// TIA Portal project "PWM TEST" (V16)

(* hardware
DEVICE "S7-1200 station_1"  S7-1200 Station
   slot 0: "Rack_0"  S7-1200 Rack  Rack  V1.0
   slot 1: "PLC_1"  CPU 1214C DC/DC/DC  6ES7 214-1AG40-0XB0  V4.2
   slot 2: "AI 4x13BIT/AQ 2x14BIT_1"  6ES7 234-4HE32-0XB0  V2.1
DEVICE "HMI_1"  KTP1200 Basic DP
   slot 0: "HMI_1"  KTP1200 Basic DP  6AV2 123-2MA03-0AX0  16.0.0.0
   slot 1: "HMI_RT_1"  KTP1200 Basic DP  6AV2 123-2MA03-0AX0  16.0.0.0
   slot 7: "HMI_1.MPI/DP_CP_1"  MPI/DP Interface  16.0.0.0
*)

// ===== PLC "PLC_1"  CPU 1214C DC/DC/DC =====

VAR_GLOBAL   // PLC tag table "Default tag table"
   "SENSOR_TOP" AT %IW64 : Int;
   "SENSOR BOTTOM" AT %IW66 : Int;
   "PUMP_PWM" AT %QW98 : Int;
   "Tag_1" AT %MD4 : Real;
   "SET POINT TANK2" AT %MW12 : Int;
   "Tag_4" AT %MD6 : Real;
   "SENSOR_CENTIMETER 2" AT %MW10 : Int;
   "Tag_5" AT %MD14 : Real;
   "SENSOR_CENTIMETER 1" AT %MW16 : Int;
   "DATA MV TANK 2" AT %MD18 : Real;
   "Tag_7" AT %MW20 : Int;
END_VAR

DATA_BLOCK "Data_TCP"   // DB2
{ S7_Optimized_Access := 'FALSE' }
VERSION : 0.1
   VAR
      DATA : Array[0..5] of Int;
   END_VAR
BEGIN
END_DATA_BLOCK

DATA_BLOCK "MB_Config"   // DB3
{ S7_Optimized_Access := 'FALSE' }
VERSION : 0.1
   VAR
      CONNECT : TCON_IP_v4;
      NDR : Bool;
      DR : Bool;
      ERROR : Bool;
      STATUS : Word;
   END_VAR
BEGIN
   CONNECT.InterfaceId := 64;
   CONNECT.ID := 1;
   CONNECT.ConnectionType := 11;
   CONNECT.RemoteAddress.ADDR[1] := 192;
   CONNECT.RemoteAddress.ADDR[2] := 168;
   CONNECT.RemoteAddress.ADDR[3] := 0;
   CONNECT.RemoteAddress.ADDR[4] := 100;
   CONNECT.LocalPort := 502;
END_DATA_BLOCK

DATA_BLOCK "DATA PID"   // DB6
{ S7_Optimized_Access := 'TRUE' }
VERSION : 0.1
   VAR
      "SP TANK2" : Real;
      "MV TANK2" : Real;
      "MV TANK2 Conv" : Real;
   END_VAR
BEGIN
END_DATA_BLOCK

FUNCTION "Scale" : Void   // FC1, LAD
{ S7_Optimized_Access := 'TRUE' }
VERSION : 0.1
BEGIN

REGION Network 1: SECSOR TANK 1
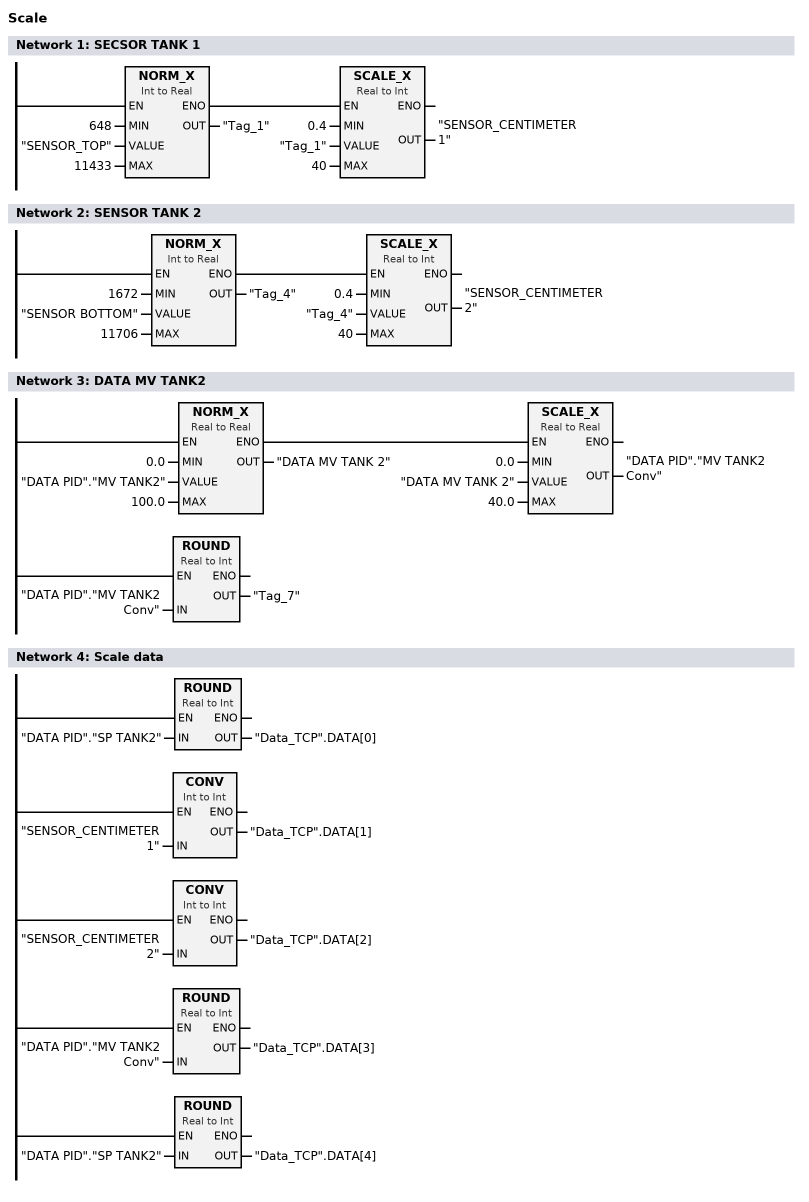
   RUNG wire#powerrail
      { S7_Templates := "[SrcType := Int, DestType := Real]" } Normalize(min := 648, value := "SENSOR_TOP", max := 11433, out => "Tag_1")
      { S7_Templates := "[SrcType := Real, DestType := Int]" } Scale(min := 0.4, value := "Tag_1", max := 40, out => "SENSOR_CENTIMETER 1")
   END_RUNG
   // the same network as SCL:
   "Tag_1" := NORM_X(MIN := 648, VALUE := "SENSOR_TOP", MAX := 11433);
   "SENSOR_CENTIMETER 1" := SCALE_X(MIN := 0.4, VALUE := "Tag_1", MAX := 40);
END_REGION

REGION Network 2: SENSOR TANK 2
   RUNG wire#powerrail
      { S7_Templates := "[SrcType := Int, DestType := Real]" } Normalize(min := 1672, value := "SENSOR BOTTOM", max := 11706, out => "Tag_4")
      { S7_Templates := "[SrcType := Real, DestType := Int]" } Scale(min := 0.4, value := "Tag_4", max := 40, out => "SENSOR_CENTIMETER 2")
   END_RUNG
   // the same network as SCL:
   "Tag_4" := NORM_X(MIN := 1672, VALUE := "SENSOR BOTTOM", MAX := 11706);
   "SENSOR_CENTIMETER 2" := SCALE_X(MIN := 0.4, VALUE := "Tag_4", MAX := 40);
END_REGION

REGION Network 3: DATA MV TANK2
   RUNG wire#powerrail
      { S7_Templates := "[SrcType := Real, DestType := Real]" } Normalize(min := 0.0, value := "DATA PID"."MV TANK2", max := 100.0, out => "DATA MV TANK 2")
      { S7_Templates := "[SrcType := Real, DestType := Real]" } Scale(min := 0.0, value := "DATA MV TANK 2", max := 40.0, out => "DATA PID"."MV TANK2 Conv")
   END_RUNG
   RUNG wire#powerrail
      { S7_Templates := "[SrcType := Real, DestType := Int]" } Round(in := "DATA PID"."MV TANK2 Conv", out => "Tag_7")
   END_RUNG
   // the same network as SCL:
   "DATA MV TANK 2" := NORM_X(MIN := 0.0, VALUE := "DATA PID"."MV TANK2", MAX := 100.0);
   "DATA PID"."MV TANK2 Conv" := SCALE_X(MIN := 0.0, VALUE := "DATA MV TANK 2", MAX := 40.0);
   "Tag_7" := ROUND("DATA PID"."MV TANK2 Conv");
END_REGION

REGION Network 4: Scale data
   RUNG wire#powerrail
      { S7_Templates := "[SrcType := Real, DestType := Int]" } Round(in := "DATA PID"."SP TANK2", out => "Data_TCP".DATA[0])
   END_RUNG
   RUNG wire#powerrail
      { S7_Templates := "[SrcType := Int, DestType := Int]" } Convert(in := "SENSOR_CENTIMETER 1", out => "Data_TCP".DATA[1])
   END_RUNG
   RUNG wire#powerrail
      { S7_Templates := "[SrcType := Int, DestType := Int]" } Convert(in := "SENSOR_CENTIMETER 2", out => "Data_TCP".DATA[2])
   END_RUNG
   RUNG wire#powerrail
      { S7_Templates := "[SrcType := Real, DestType := Int]" } Round(in := "DATA PID"."MV TANK2 Conv", out => "Data_TCP".DATA[3])
   END_RUNG
   RUNG wire#powerrail
      { S7_Templates := "[SrcType := Real, DestType := Int]" } Round(in := "DATA PID"."SP TANK2", out => "Data_TCP".DATA[4])
   END_RUNG
   // the same network as SCL:
   "Data_TCP".DATA[0] := ROUND("DATA PID"."SP TANK2");
   "Data_TCP".DATA[1] := INT_TO_INT("SENSOR_CENTIMETER 1");
   "Data_TCP".DATA[2] := INT_TO_INT("SENSOR_CENTIMETER 2");
   "Data_TCP".DATA[3] := ROUND("DATA PID"."MV TANK2 Conv");
   "Data_TCP".DATA[4] := ROUND("DATA PID"."SP TANK2");
END_REGION
END_FUNCTION

ORGANIZATION_BLOCK "Main"   // OB1, LAD, ProgramCycle
TITLE = "Main Program Sweep (Cycle)"
{ S7_Optimized_Access := 'TRUE' }
VERSION : 0.1
   VAR_INPUT
      Initial_Call : Bool;   // Initial call of this OB
      Remanence : Bool;   // =True, if remanent data are available
   END_VAR
BEGIN

REGION Network 1: SETPOINT
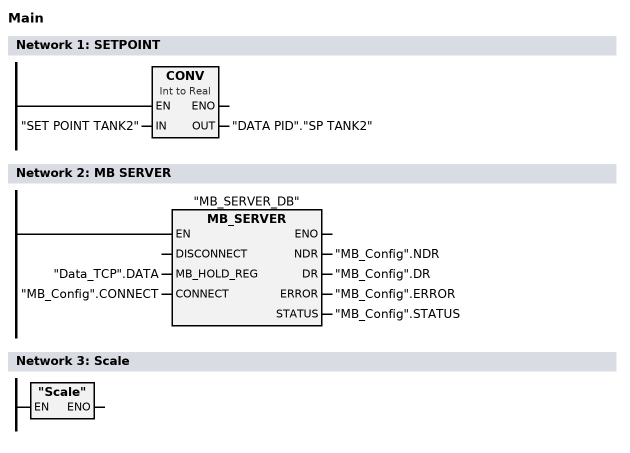
   RUNG wire#powerrail
      { S7_Templates := "[SrcType := Int, DestType := Real]" } Convert(in := "SET POINT TANK2", out => "DATA PID"."SP TANK2")
   END_RUNG
   // the same network as SCL:
   "DATA PID"."SP TANK2" := INT_TO_REAL("SET POINT TANK2");
END_REGION

REGION Network 2: MB SERVER
   "MB_SERVER_DB"(MB_HOLD_REG := "Data_TCP".DATA,   // MB_SERVER
                  CONNECT := "MB_Config".CONNECT,
                  NDR => "MB_Config".NDR,
                  DR => "MB_Config".DR,
                  ERROR => "MB_Config".ERROR,
                  STATUS => "MB_Config".STATUS);
END_REGION

REGION Network 3: Scale
   RUNG wire#powerrail
      "Scale"()
   END_RUNG
   // the same network as SCL:
   "Scale"();
END_REGION
END_ORGANIZATION_BLOCK

ORGANIZATION_BLOCK "Cyclic interrupt"   // OB30, LAD, CyclicInterrupt
{ S7_Optimized_Access := 'TRUE' }
VERSION : 0.1
   VAR_INPUT
      Initial_Call : Bool;   // Initial call of this OB
      Event_Count : Int;   // Events discarded
   END_VAR
BEGIN

REGION Network 1
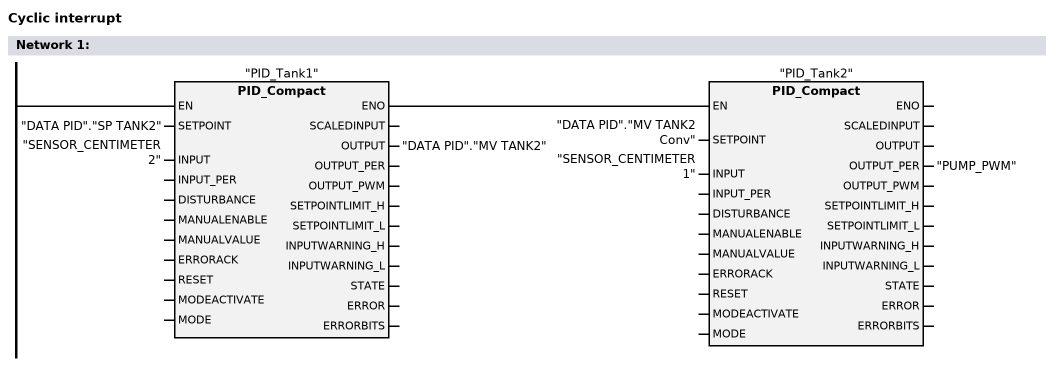
   // ENO of a box is taken as its EN; it also drops when the box reports an error
   "PID_Tank1"(Setpoint := "DATA PID"."SP TANK2",   // PID_Compact
               Input := "SENSOR_CENTIMETER 2",
               Output => "DATA PID"."MV TANK2");
   "PID_Tank2"(Setpoint := "DATA PID"."MV TANK2 Conv", Input := "SENSOR_CENTIMETER 1", Output_PER => "PUMP_PWM");   // PID_Compact
END_REGION
END_ORGANIZATION_BLOCK

(* ===== HMI "HMI_RT_1" =====
system functions are stored by id; their names below are inferred from use

HMI tags "Default tag table"
   "Tag_ScreenNumber" : UInt, internal

Template "Template_1" 1280x800
   Button "Exit" at 1182,752 size 67x47; TextOff 'Exit'; PictureOff "ExitRuntime_KTP1200_Basic_DP_TR"; PictureOn "ExitRuntime_KTP1200_Basic_DP_TR"
      on Release: StopRuntime(0)
   Button "Template_Button" at 1054,752 size 67x47; TextOff 'Text'
   Button "Template_Button_1" at 926,752 size 67x47; TextOff 'Text'
   Button "Template_Button_2" at 798,752 size 67x47; TextOff 'Text'
   Button "Template_Button_3" at 670,752 size 67x47; TextOff 'Text'
   Button "Template_Button_4" at 542,752 size 67x47; TextOff 'Text'
   Button "Template_Button_5" at 414,752 size 67x47; TextOff 'Text'
   Button "Template_Button_6" at 286,752 size 67x47; TextOff 'Text'
   Button "Alarms" at 158,752 size 67x47; TextOff 'Alarms'; PictureOff "AlarmDisplay_KTP1200_Basic_DP_TR"; PictureOn "AlarmDisplay_KTP1200_Basic_DP_TR"
      on Release: function_ef3f5d25("Alarm window_Unacknowledged", -1)
   Button "Start screen" at 30,752 size 67x47; TextOff 'Start screen'; PictureOff "NavigateHome_KTP1200_Basic_DP_TR"; PictureOn "NavigateHome_KTP1200_Basic_DP_TR"
      on Release: ActivateScreen("Root screen", 0)
   SymbolicIOField "Symbolic_IO_Field_Screen" at 87,9 size 1086x30; TextOff '0'; TextOn '1'; TextList "TextList_ScreenNames"
      ProcessValue <- "Tag_ScreenNumber"
      on Change: ActivateScreenByNumber("Tag_ScreenNumber", 0)
   DateTimeField "HmiScreenItemData" at 1175,24 size 105x24
   DateTimeField "HmiScreenItemData_1" at 1175,0 size 105x24
   GraphicView "Logo" at 0,0 size 85x48; Picture "Logo of HMI_1"

screen "Root screen" 1280x800, template "Template_1"
   on GenerateScreen: SetTag("Tag_ScreenNumber", 1)
*)